// TIA Portal V17 export
// export: Created 2025-03-07T09:24:05.4702193Z, ExportSetting WithDefaults, DisplayName Totally Integrated Automation Portal, DisplayVersion V17 Update 8, DisplayName TIA Portal Openness, DisplayVersion V17 Update 8, DisplayName TIA Portal Version Control Interface, DisplayVersion V17, DisplayName SINAMICS Startdrive Advanced, DisplayVersion V17 SP2, DisplayName SINAMICS Startdrive G110M, G120, G120C, G120D, G120P, G115D, DisplayVersion V17 SP2, DisplayName SINAMICS Startdrive G130, G150, S120, S150, SINAMICS MV, S210, DisplayVersion V17 SP2, DisplayName STEP 7 Professional, DisplayVersion V17 Update 8, DisplayName SINUMERIK ONE STEP 7 Toolbox, DisplayVersion V17 Update 12, DisplayName SINUMERIK 840D sl STEP 7 Toolbox, DisplayVersion V17 Update 12, DisplayName STEP 7 Safety, DisplayVersion V17 Update 6, DisplayName WinCC Advanced, DisplayVersion V17 Update 8
FUNCTION "FC22000_HOPPER_SYSTEM_MAIN" : Void   // FC22000, LAD
TITLE = FC22000 HOPPER SYSTEM MAIN
{ S7_Optimized_Access := 'TRUE' }
VERSION : 0.1
// stored: AutoNumber false, IsIECCheckEnabled false, SetENOAutomatically false, UDAEnableTagReadback false
BEGIN

REGION Network 1: FC22100_HOPPER_SYSTEM_SENSORS
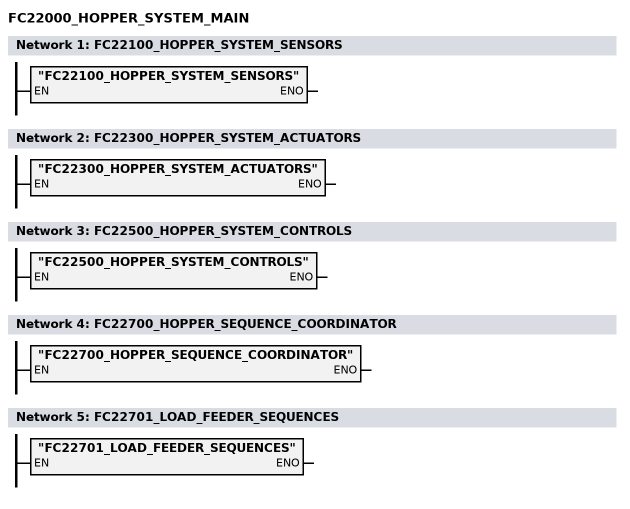
   RUNG wire#powerrail
      "FC22100_HOPPER_SYSTEM_SENSORS"()
   END_RUNG
   // the same network as SCL:
   "FC22100_HOPPER_SYSTEM_SENSORS"();
END_REGION

REGION Network 2: FC22300_HOPPER_SYSTEM_ACTUATORS
   RUNG wire#powerrail
      "FC22300_HOPPER_SYSTEM_ACTUATORS"()
   END_RUNG
   // the same network as SCL:
   "FC22300_HOPPER_SYSTEM_ACTUATORS"();
END_REGION

REGION Network 3: FC22500_HOPPER_SYSTEM_CONTROLS
   RUNG wire#powerrail
      "FC22500_HOPPER_SYSTEM_CONTROLS"()
   END_RUNG
   // the same network as SCL:
   "FC22500_HOPPER_SYSTEM_CONTROLS"();
END_REGION

REGION Network 4: FC22700_HOPPER_SEQUENCE_COORDINATOR
   RUNG wire#powerrail
      "FC22700_HOPPER_SEQUENCE_COORDINATOR"()
   END_RUNG
   // the same network as SCL:
   "FC22700_HOPPER_SEQUENCE_COORDINATOR"();
END_REGION

REGION Network 5: FC22701_LOAD_FEEDER_SEQUENCES
   RUNG wire#powerrail
      "FC22701_LOAD_FEEDER_SEQUENCES"()
   END_RUNG
   // the same network as SCL:
   "FC22701_LOAD_FEEDER_SEQUENCES"();
END_REGION
END_FUNCTION
